FUNCTION_BLOCK FB_Test
VAR
	nCounter : LINT;
END_VAR

nCounter := nCounter +1;

END_FUNCTION_BLOCK

(* stored: Version 1.1.0.1, ProductVersion 3.1.4024.12
   POU FB_Test: Id {5b98af6c-bc09-4483-93a2-391d8cb1c473}, SpecialFunc None *)
